PROGRAM prgCom
VAR
	fbCom			: FB_MqttCommunicator_V3;
END_VAR

fbCom(
	bConnect:= TRUE, 
	strAuthKey := 'TSG88376368072',
	sUserName:= '4e725250-0700-401c-9007-6635df778dc6', 
	sUserPassword:= 'e61f3a0f-7441-47a1-b0d1-b48ec32b2934', 
	eSavePositionCertificate:= eSavePositionOnPLC.ePostionC,
	bConnected=> , 
	bError=> , 
	hrErrorCode=> , 
	eConnectionState=> , 
	eErrorMessage_Out=> );

END_PROGRAM

(* stored: Version 1.1.0.1, ProductVersion 3.1.4024.12
   POU prgCom: Id {ab2e2113-e5ef-4576-b3e1-d9e4709b48fc}, SpecialFunc None *)
